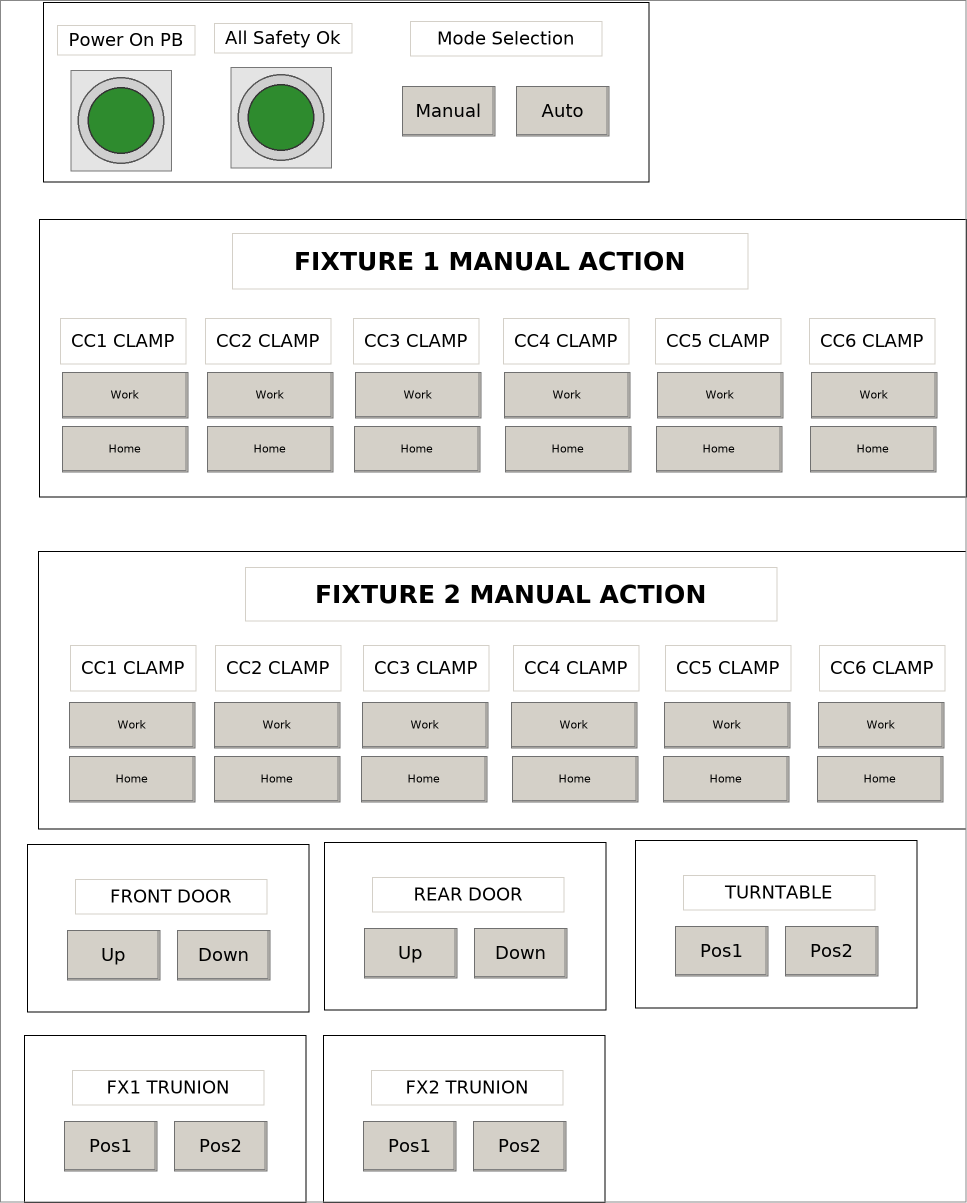
VISUALIZATION Fixture_Manual  // 967x1203
    Rectangle (27,844 282x168)
    Rectangle (38,551 928x278)
    Rectangle (39,219 928x278)
    Rectangle (43,2 606x180)
    Textfield (232,233 516x56), "FIXTURE 1 MANUAL ACTION"
    Button (62,372 126x46), "Work", colour toggle: Inputs.i_FX1_CC1_Clamp_1_Sensor_WP
        tap Memory_DB.M_FX1_CC1_CLAMPING_UNIT1_3_WP
    Button (62,426 126x46), "Home", colour toggle: Inputs.i_FX1_CC1_Clamp_1_Sensor_HP
        tap Memory_DB.M_FX1_CC1_CLAMPING_UNIT1_3_HP
    Textfield (60,318 126x46), "CC1 CLAMP"
    Button (355,372 126x46), "Work", colour toggle: Inputs.i_FX1_CC3_Clamp_1_Sensor_WP
        tap Memory_DB.M_FX1_CC3_CLAMPING_UNIT3_3_WP
    Button (354,426 126x46), "Home", colour toggle: Inputs.i_FX1_CC3_Clamp_1_Sensor_HP
        tap Memory_DB.M_FX1_CC3_CLAMPING_UNIT3_3_HP
    Button (504,372 126x46), "Work", colour toggle: Inputs.i_FX1_CC4_Clamp_1_Sensor_WP
        tap Memory_DB.M_FX1_CC4_CLAMPING_UNIT4_3_WP
    Button (505,426 126x46), "Home", colour toggle: Inputs.i_FX1_CC4_Clamp_1_Sensor_HP
        tap Memory_DB.M_FX1_CC4_CLAMPING_UNIT4_3_HP
    Button (657,372 126x46), "Work", colour toggle: Inputs.i_FX1_CC5_Clamp_1_Sensor_WP
        tap Memory_DB.M_FX1_CC5_CLAMPING_UNIT5_1_WP
    Button (656,426 126x46), "Home", colour toggle: Inputs.i_FX1_CC5_Clamp_1_Sensor_HP
        tap Memory_DB.M_FX1_CC5_CLAMPING_UNIT5_1_HP
    Button (811,372 126x46), "Work", colour toggle: Inputs.i_FX1_CC6_Clamp_1_Sensor_WP
        tap Memory_DB.M_FX1_CC6_CLAMPING_UNIT6_1_WP
    Button (810,426 126x46), "Home", colour toggle: Inputs.i_FX1_CC6_Clamp_1_Sensor_HP
        tap Memory_DB.M_FX1_CC6_CLAMPING_UNIT6_1_hP
    Button (207,372 126x46), "Work", colour toggle: Inputs.i_FX1_CC2_Clamp_1_Sensor_WP
        tap Memory_DB.M_FX1_CC2_CLAMPING_UNIT2_3_WP
    Button (207,426 126x46), "Home", colour toggle: Inputs.i_FX1_CC2_Clamp_1_Sensor_HP
        tap Memory_DB.M_FX1_CC2_CLAMPING_UNIT2_3_HP
    Textfield (503,318 126x46), "CC4 CLAMP"
    Textfield (655,318 126x46), "CC5 CLAMP"
    Textfield (809,318 126x46), "CC6 CLAMP"
    Textfield (205,318 126x46), "CC2 CLAMP"
    Textfield (353,318 126x46), "CC3 CLAMP"
    Textfield (245,567 532x54), "FIXTURE 2 MANUAL ACTION"
    Textfield (70,645 126x46), "CC1 CLAMP"
    Textfield (513,645 126x46), "CC4 CLAMP"
    Textfield (665,645 126x46), "CC5 CLAMP"
    Textfield (819,645 126x46), "CC6 CLAMP"
    Textfield (215,645 126x46), "CC2 CLAMP"
    Textfield (363,645 126x46), "CC3 CLAMP"
    PushSwitch (66,70 110x101), variable: Inputs.i_Power_On_PB, behaviour: TOGGLE, style: Switch-PushSwitch-Green
    Textfield (57,25 138x30), "Power On PB"
    PushSwitch (226,67 110x101), variable: Memory_DB.M_Safety_Ok, behaviour: TOGGLE, style: Switch-PushSwitch-Green
    Textfield (214,23 138x30), "All Safety Ok"
    Button (402,86 93x50), "Manual", text variable: Inputs.i_Mode_Select, colour toggle: Memory_DB.M_Manual_Active
        OnMouseClick: write the text variable via VisuDialogs.Numpad
    Textfield (410,21 192x35), "Mode Selection"
    Button (516,86 93x50), "Auto", text variable: Inputs.i_Mode_Select, colour toggle: Memory_DB.M_Auto_Active
        OnMouseClick: write the text variable via VisuDialogs.Numpad
    Button (69,702 126x46), "Work", colour toggle: Inputs.i_FX2_CC1_Clamp_1_Sensor_WP
        tap Memory_DB.M_FX2_CC1_CLAMPING_UNIT1_3_WP
    Button (69,756 126x46), "Home", colour toggle: Inputs.i_FX2_CC1_Clamp_1_Sensor_HP
        tap Memory_DB.M_FX2_CC1_CLAMPING_UNIT1_3_HP
    Button (362,702 126x46), "Work", colour toggle: Inputs.i_FX2_CC3_Clamp_1_Sensor_WP
        tap Memory_DB.M_FX2_CC3_CLAMPING_UNIT3_3_WP
    Button (361,756 126x46), "Home", colour toggle: Inputs.i_FX2_CC3_Clamp_1_Sensor_HP
        tap Memory_DB.M_FX2_CC3_CLAMPING_UNIT3_3_HP
    Button (511,702 126x46), "Work", colour toggle: Inputs.i_FX2_CC4_Clamp_1_Sensor_WP
        tap Memory_DB.M_FX2_CC4_CLAMPING_UNIT4_3_WP
    Button (512,756 126x46), "Home", colour toggle: Inputs.i_FX2_CC4_Clamp_1_Sensor_HP
        tap Memory_DB.M_FX2_CC4_CLAMPING_UNIT4_3_HP
    Button (664,702 126x46), "Work", colour toggle: Inputs.i_FX2_CC5_Clamp_1_Sensor_WP
        tap Memory_DB.M_FX2_CC5_CLAMPING_UNIT5_1_WP
    Button (663,756 126x46), "Home", colour toggle: Inputs.i_FX2_CC5_Clamp_1_Sensor_HP
        tap Memory_DB.M_FX2_CC5_CLAMPING_UNIT5_1_HP
    Button (818,702 126x46), "Work", colour toggle: Inputs.i_FX2_CC6_Clamp_1_Sensor_WP
        tap Memory_DB.M_FX2_CC6_CLAMPING_UNIT6_1_WP
    Button (817,756 126x46), "Home", colour toggle: Inputs.i_FX2_CC6_Clamp_1_Sensor_HP
        tap Memory_DB.M_FX2_CC6_CLAMPING_UNIT6_1_hP
    Button (214,702 126x46), "Work", colour toggle: Inputs.i_FX2_CC2_Clamp_1_Sensor_WP
        tap Memory_DB.M_FX2_CC2_CLAMPING_UNIT2_3_WP
    Button (214,756 126x46), "Home", colour toggle: Inputs.i_FX2_CC2_Clamp_1_Sensor_HP
        tap Memory_DB.M_FX2_CC2_CLAMPING_UNIT2_3_HP
    Textfield (75,879 192x35), "FRONT DOOR"
    Button (67,930 93x50), "Up", text variable: Inputs.i_Mode_Select, colour toggle: Inputs.i_Front_Door_Up
        tap Memory_DB.M_FRONT_DOOR_UP
    Button (177,930 93x50), "Down", text variable: Inputs.i_Mode_Select, colour toggle: Inputs.i_Front_Door_Down
        tap Memory_DB.M_FRONT_DOOR_DOWN
    Rectangle (324,842 282x168)
    Textfield (372,877 192x35), "REAR DOOR"
    Button (364,928 93x50), "Up", text variable: Inputs.i_Mode_Select, colour toggle: Inputs.i_Rear_Door_Up
        tap Memory_DB.M_REAR_DOOR_UP
    Button (474,928 93x50), "Down", text variable: Inputs.i_Mode_Select, colour toggle: Inputs.i_Rear_Door_Down
        tap Memory_DB.M_REAR_DOOR_DOWN
    Rectangle (635,840 282x168)
    Textfield (683,875 192x35), "TURNTABLE"
    Button (675,926 93x50), "Pos1", text variable: Inputs.i_Mode_Select, colour toggle: Memory_DB.M_Turntable_POS1_Reached
        tap Memory_DB.M_Turntable_POS1_CMD
    Button (785,926 93x50), "Pos2", text variable: Inputs.i_Mode_Select, colour toggle: Memory_DB.M_Turntable_POS2_Reached
        tap Memory_DB.M_Turntable_POS2_CMD
    Rectangle (24,1035 282x168)
    Textfield (72,1070 192x35), "FX1 TRUNION"
    Button (64,1121 93x50), "Pos1", text variable: Inputs.i_Mode_Select, colour toggle: Memory_DB.M_Fixture1_TR_POS1_Reached
        tap Memory_DB.M_Fixture1_TR_POS1_CMD
    Button (174,1121 93x50), "Pos2", text variable: Inputs.i_Mode_Select, colour toggle: Memory_DB.M_Fixture1_TR_POS2_Reached
        tap Memory_DB.M_Fixture1_TR_POS2_CMD
    Rectangle (323,1035 282x168)
    Textfield (371,1070 192x35), "FX2 TRUNION"
    Button (363,1121 93x50), "Pos1", text variable: Inputs.i_Mode_Select, colour toggle: Memory_DB.M_Fixture2_TR_POS1_Reached
        tap Memory_DB.M_Fixture2_TR_POS1_CMD
    Button (473,1121 93x50), "Pos2", text variable: Inputs.i_Mode_Select, colour toggle: Memory_DB.M_Fixture2_TR_POS2_Reached
        tap Memory_DB.M_Fixture2_TR_POS2_CMD
END_VISUALIZATION

(* stored: Version 1.1.0.1, ProductVersion 3.1.4024.16
   Visu Fixture_Manual: Id {8370cfdf-5888-4612-b097-fdda834b135d} *)
